// TIA Portal V16 program export: 1 tag tables, 0 data types, 1 data blocks, 4 code blocks (in call order from the OBs), 0 instance data blocks

VAR_GLOBAL   // PLC tag table "Tabla de variables estándar"
   System_Byte AT %MB1 : Byte;
   FirstScan AT %M1.0 : Bool;
   DiagStatusUpdate AT %M1.1 : Bool;
   AlwaysTRUE AT %M1.2 : Bool;
   AlwaysFALSE AT %M1.3 : Bool;
   Clock_Byte AT %MB0 : Byte;
   Clock_10Hz AT %M0.0 : Bool;
   Clock_5Hz AT %M0.1 : Bool;
   "Clock_2.5Hz" AT %M0.2 : Bool;
   Clock_2Hz AT %M0.3 : Bool;
   "Clock_1.25Hz" AT %M0.4 : Bool;
   Clock_1Hz AT %M0.5 : Bool;
   "Clock_0.625Hz" AT %M0.6 : Bool;
   "Clock_0.5Hz" AT %M0.7 : Bool;
   G120_VActual AT %IW62 : Int;
   VActual_Escalada AT %MD60 : Real;
   Setpoint_Escalado AT %MD64 : Real;
   G120_Setpoint AT %QW62 : Int;
   SensorT AT %IW64 : Int;
   SensorN AT %IW66 : Int;
END_VAR

DATA_BLOCK "Analogicas"   // DB1
{ S7_Optimized_Access := 'TRUE' }
VERSION : 0.1
// stored: AutoNumber true, DBAccessibleFromOPCUA true, IsOnlyStoredInLoadMemory false, IsRetainMemResEnabled false, IsWriteProtectedInAS false, MemoryReserve 100
   VAR
      Temperatura : Struct
         Lubricador1 : Real;
         Horno2 : Real;
      END_STRUCT;
      Nivel : Struct
         Tanque3 : Real;
         Silo4 : Real;
      END_STRUCT;
      Presion : Struct
         Impulsion5 : Real;
         Rebombeo6 : Real;
      END_STRUCT;
   END_VAR
BEGIN
END_DATA_BLOCK

ORGANIZATION_BLOCK "Main"   // OB1, LAD, ProgramCycle
TITLE = "Main Program Sweep (Cycle)"
{ S7_Optimized_Access := 'TRUE' }
VERSION : 0.1
// stored: AutoNumber true, IsIECCheckEnabled false, SetENOAutomatically false
   VAR_INPUT
      Initial_Call : Bool;   // Initial call of this OB
      Remanence : Bool;   // =True, if remanent data are available
   END_VAR
BEGIN

REGION Network 1
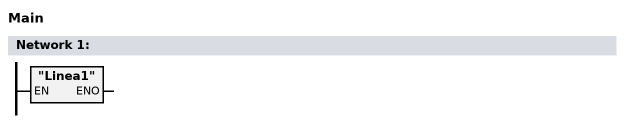
   RUNG wire#powerrail
      "Linea1"()
   END_RUNG
   // the same network as SCL:
   "Linea1"();
END_REGION
END_ORGANIZATION_BLOCK

FUNCTION "Linea1" : Void   // FC2, LAD
{ S7_Optimized_Access := 'TRUE' }
VERSION : 0.1
// stored: AutoNumber true, IsIECCheckEnabled false, SetENOAutomatically false, UDAEnableTagReadback false
BEGIN

REGION Network 1
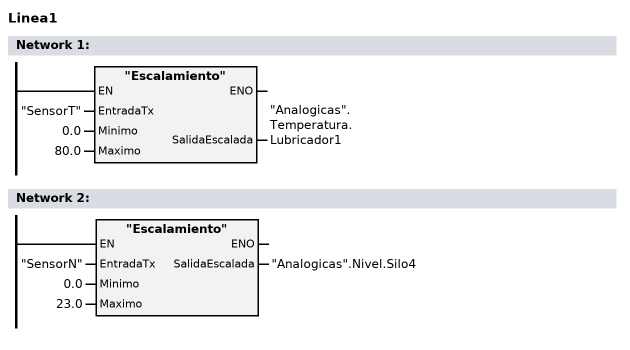
   RUNG wire#powerrail
      "Escalamiento"(EntradaTx := "SensorT", Minimo := 0.0, Maximo := 80.0, SalidaEscalada => "Analogicas".Temperatura.Lubricador1)
   END_RUNG
   // the same network as SCL:
   "Escalamiento"(EntradaTx := "SensorT",
                  Minimo := 0.0,
                  Maximo := 80.0,
                  SalidaEscalada => "Analogicas".Temperatura.Lubricador1);
END_REGION

REGION Network 2
   RUNG wire#powerrail
      "Escalamiento"(EntradaTx := "SensorN", Minimo := 0.0, Maximo := 23.0, SalidaEscalada => "Analogicas".Nivel.Silo4)
   END_RUNG
   // the same network as SCL:
   "Escalamiento"(EntradaTx := "SensorN",
                  Minimo := 0.0,
                  Maximo := 23.0,
                  SalidaEscalada => "Analogicas".Nivel.Silo4);
END_REGION
END_FUNCTION

FUNCTION "Escalamiento" : Void   // FC1, LAD
{ S7_Optimized_Access := 'TRUE' }
VERSION : 0.1
// stored: AutoNumber true, IsIECCheckEnabled false, SetENOAutomatically false, UDAEnableTagReadback false
   VAR_INPUT
      EntradaTx : Int;
      Minimo : Real;
      Maximo : Real;
   END_VAR
   VAR_OUTPUT
      SalidaEscalada : Real;
   END_VAR
   VAR_TEMP
      entrada_norm : Real;
   END_VAR
BEGIN

REGION Network 1
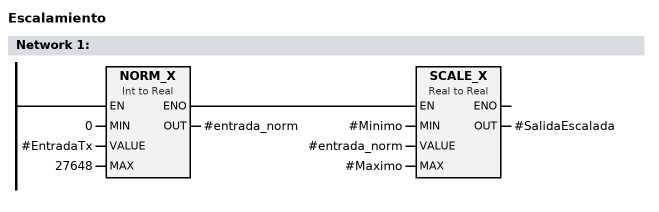
   RUNG wire#powerrail
      { S7_Templates := "[SrcType := Int, DestType := Real]" } Normalize(min := 0, value := #EntradaTx, max := 27648, out => #entrada_norm)
      { S7_Templates := "[SrcType := Real, DestType := Real]" } Scale(min := #Minimo, value := #entrada_norm, max := #Maximo, out => #SalidaEscalada)
   END_RUNG
   // the same network as SCL:
   #entrada_norm := NORM_X(MIN := 0, VALUE := #EntradaTx, MAX := 27648);
   #SalidaEscalada := SCALE_X(MIN := #Minimo, VALUE := #entrada_norm, MAX := #Maximo);
END_REGION
END_FUNCTION

FUNCTION "Escalamiento_G120" : Void   // FC10, LAD
{ S7_Optimized_Access := 'TRUE' }
VERSION : 0.1
// stored: AutoNumber false, IsIECCheckEnabled false, SetENOAutomatically false, UDAEnableTagReadback false
   VAR_TEMP
      vactual_norm : Real;
      setpoint_norm : Real;
   END_VAR
BEGIN

REGION Network 1: Escalar Velocidad actual
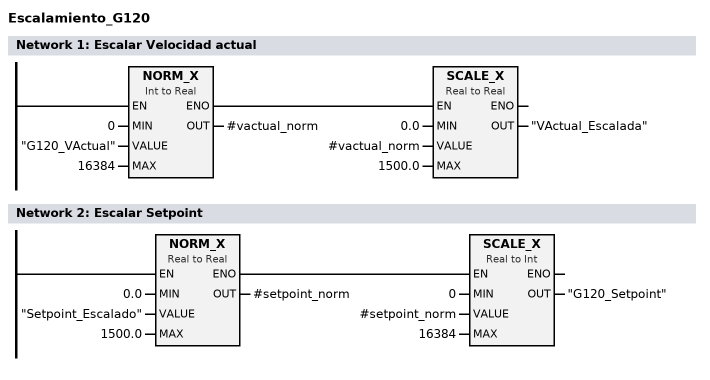
   RUNG wire#powerrail
      { S7_Templates := "[SrcType := Int, DestType := Real]" } Normalize(min := 0, value := "G120_VActual", max := 16384, out => #vactual_norm)
      { S7_Templates := "[SrcType := Real, DestType := Real]" } Scale(min := 0.0, value := #vactual_norm, max := 1500.0, out => "VActual_Escalada")
   END_RUNG
   // the same network as SCL:
   #vactual_norm := NORM_X(MIN := 0, VALUE := "G120_VActual", MAX := 16384);
   "VActual_Escalada" := SCALE_X(MIN := 0.0, VALUE := #vactual_norm, MAX := 1500.0);
END_REGION

REGION Network 2: Escalar Setpoint
   RUNG wire#powerrail
      { S7_Templates := "[SrcType := Real, DestType := Real]" } Normalize(min := 0.0, value := "Setpoint_Escalado", max := 1500.0, out => #setpoint_norm)
      { S7_Templates := "[SrcType := Real, DestType := Int]" } Scale(min := 0, value := #setpoint_norm, max := 16384, out => "G120_Setpoint")
   END_RUNG
   // the same network as SCL:
   #setpoint_norm := NORM_X(MIN := 0.0, VALUE := "Setpoint_Escalado", MAX := 1500.0);
   "G120_Setpoint" := SCALE_X(MIN := 0, VALUE := #setpoint_norm, MAX := 16384);
END_REGION
END_FUNCTION
